// TIA Portal V20 export
TYPE "typeCmHmiInterface"
// stored: Access Published, Namespace Unit1.Em8
   STRUCT
      softcam : "Unit1.Em8.typeCmHmiInterfaceSoftCam";
      brakeTest : "Unit1.Em8.typeCmHmiInterfaceBrakeTest";
   END_STRUCT;
END_TYPE
